// TIA Portal V17 export
// export: Created 2023-12-05T13:40:24.2794023Z, ExportSetting WithDefaults, DisplayName Totally Integrated Automation Portal, DisplayVersion V17, DisplayName TIA Portal Openness, DisplayVersion V17, DisplayName TIA Portal Version Control Interface, DisplayVersion V17, DisplayName SINAMICS Startdrive Advanced, DisplayVersion V17, DisplayName SINAMICS Startdrive G130, G150, S120, S150, SINAMICS MV, S210, DisplayVersion V17, DisplayName SINAMICS Startdrive G110M, G120, G120C, G120D, G120P, G115D, DisplayVersion V17, DisplayName STEP 7 Professional, DisplayVersion V17, DisplayName STEP 7 Safety, DisplayVersion V17, DisplayName WinCC Professional, DisplayVersion V17
DATA_BLOCK "KNIFE_AND_SLUG_COUNTERS"   // DB402
{ S7_Optimized_Access := 'FALSE' }
VERSION : 0.1
// stored: AutoNumber false, DBAccessibleFromOPCUA true, DBAccessibleFromWebserver true, IsOnlyStoredInLoadMemory false, IsWriteProtectedInAS false
   VAR RETAIN
      ST1OP02 { S7_SetPoint := 'True'} : "Counter Knife";
      ST1OP03 { S7_SetPoint := 'True'} : "Counter Knife";
      ST2OP18 { S7_SetPoint := 'True'} : "Counter Knife";
      ST1OP02_Box { S7_SetPoint := 'True'} : "Slug counter";
      ST1OP03_Box { S7_SetPoint := 'True'} : "Slug counter";
      ST2OP18_Box { S7_SetPoint := 'True'} : "Slug counter";
   END_VAR
BEGIN
   ST1OP02.Counter_changeKnife.Work_Bit1 := FALSE;
   ST1OP02.Counter_changeKnife.Work_Bit2 := FALSE;
   ST1OP02.Counter_changeKnife.reset := FALSE;
   ST1OP02.Counter_changeKnife.Count_DOWN := 30000;
   ST1OP02.Counter_changeKnife.value := 30000;
   ST1OP03.Counter_changeKnife.Work_Bit1 := FALSE;
   ST1OP03.Counter_changeKnife.Work_Bit2 := FALSE;
   ST1OP03.Counter_changeKnife.reset := FALSE;
   ST1OP03.Counter_changeKnife.Count_DOWN := 30000;
   ST1OP03.Counter_changeKnife.value := 30000;
   ST2OP18.Counter_changeKnife.Work_Bit1 := FALSE;
   ST2OP18.Counter_changeKnife.Work_Bit2 := FALSE;
   ST2OP18.Counter_changeKnife.reset := FALSE;
   ST2OP18.Counter_changeKnife.Count_DOWN := 30000;
   ST2OP18.Counter_changeKnife.value := 30000;
   ST1OP02_Box.Counter_slug.Work_Bit1 := FALSE;
   ST1OP02_Box.Counter_slug.Work_Bit2 := TRUE;
   ST1OP02_Box.Counter_slug.reset := TRUE;
   ST1OP02_Box.Counter_slug.Count_DOWN := 1000;
   ST1OP02_Box.Counter_slug.value := 1000;
   ST1OP03_Box.Counter_slug.Work_Bit1 := FALSE;
   ST1OP03_Box.Counter_slug.Work_Bit2 := FALSE;
   ST1OP03_Box.Counter_slug.reset := FALSE;
   ST1OP03_Box.Counter_slug.Count_DOWN := 1000;
   ST1OP03_Box.Counter_slug.value := 1000;
   ST2OP18_Box.Counter_slug.Work_Bit1 := FALSE;
   ST2OP18_Box.Counter_slug.Work_Bit2 := TRUE;
   ST2OP18_Box.Counter_slug.reset := TRUE;
   ST2OP18_Box.Counter_slug.Count_DOWN := 4000;
   ST2OP18_Box.Counter_slug.value := 4000;
END_DATA_BLOCK
